# EPICS substitutions: ISIS/lvexportApp/Db/user.substitutions
# Example substitutions file

file "db/dbExample1.db" {
    { user = "faa59" }
}

file db/dbExample2.db {
    pattern { user, no, scan }
        { "faa59", 1, "1 second" }
        { "faa59", 2, "2 second" }
        { "faa59", 3, "5 second" }
}
